Yaskawa INFORM job: R1_W26(-90,90)(KAMERA).JBI

/JOB
//NAME R1_W26(-90,90)(KAMERA)
//POS
///NPOS 78,78,0,7,0,0
///TOOL 0
///POSTYPE PULSE
///PULSE
C00000=-75114,-71893,-86548,-16593,83246,79420
C00001=-80306,-57562,-63247,-15413,75536,78631
C00002=-81645,-55087,-59639,-15080,74370,78302
C00003=-81645,-55006,-58527,-15126,73749,78382
C00004=-81645,-55025,-58760,-15117,73878,78365
C00005=-82615,-56005,-59303,-14838,73537,78058
C00006=-81645,-55079,-59521,-15087,74304,78310
C00007=-93593,1947,-22095,-11058,78527,73697
C00008=-93896,1420,-20145,-11015,77043,73728
C00009=-93896,1359,-19447,-11035,76591,73769
C00010=-93896,1375,-19639,-11030,76716,73757
C00011=-94601,778,-20143,-10801,76623,73523
C00012=-93896,1456,-20502,-11006,77276,73706
C00013=-99701,55982,31111,-9246,72874,72061
C00014=-100041,56496,33717,-9193,71511,72046
C00015=-100041,56569,34702,-9223,70950,72089
C00016=-100041,56551,34487,-9216,71073,72080
C00017=-100636,55976,33841,-9009,71106,71866
C00018=-100041,56488,33604,-9190,71578,72041
C00019=-99543,52569,25332,-9219,74671,71979
C00020=-97259,35030,-12066,-9701,88745,71659
C00021=-112921,-101015,-99029,5314,69459,84771
C00022=-131689,-93265,-75977,27197,64180,77750
C00023=-125720,-68183,-62010,24523,66206,80662
C00024=-125720,-67997,-61190,24597,65833,80578
C00025=-125720,-68044,-61398,24578,65929,80599
C00026=-124863,-68129,-61441,24298,65661,80883
C00027=-125720,-68320,-62645,24468,66502,80726
C00028=-125720,-68684,-64449,24312,67343,80914
C00029=-124059,-8041,-25847,22767,73693,82865
C00030=-124059,-8098,-23570,22924,72370,82603
C00031=-124059,-8098,-23067,22960,72086,82548
C00032=-124059,-8098,-23269,22945,72201,82571
C00033=-123393,-8156,-23316,22717,72018,82785
C00034=-124059,-8088,-24456,22861,72880,82707
C00035=-124059,-8025,-26153,22747,73876,82901
C00036=-123243,49165,27702,22910,70180,82472
C00037=-123243,49353,29898,23083,69020,82237
C00038=-123243,49474,30981,23171,68462,82121
C00039=-123243,49447,30748,23151,68580,82145
C00040=-122653,49389,30685,22948,68426,82342
C00041=-123243,49309,29455,23047,69250,82282
C00042=-123261,47212,24063,22760,71328,82695
C00043=-127182,-101970,-83118,25859,62678,79240
C00044=-148123,-105377,-50787,80405,47389,50643
C00045=-144996,-106265,-51019,81268,45275,50701
C00046=-125639,-92184,-72932,25604,61069,79507
C00047=-125809,-91535,-71625,25772,60696,79344
C00048=-125196,-74812,-64441,24671,64300,80456
C00049=-124580,-57199,-55547,23834,67394,81387
C00050=-124115,-40866,-46002,23300,69579,82027
C00051=-123813,-29133,-38349,23019,70716,82374
C00052=-123561,-15314,-28491,22802,71603,82649
C00053=-123288,-2303,-18230,22666,71872,82806
C00054=-123046,12376,-5585,22611,71586,82839
C00055=-122891,24863,5995,22646,70888,82760
C00056=-122733,39263,20347,22777,69515,82548
C00057=-122600,54559,36695,23052,67446,82176
C00058=-122491,73744,58718,23649,64007,81492
C00059=-122584,71948,49831,22918,68228,82344
C00060=-109861,31401,-26015,2772,95783,84263
C00061=-100600,-80082,-88673,-18141,88148,63436
C00062=-108129,-100882,-75117,-22380,56663,65945
C00063=-110628,-101357,-75286,-21477,55869,65041
C00064=-108411,-101318,-76207,-22166,57003,65749
C00065=-110367,-78057,-70654,-16601,76479,61655
C00066=-111567,-60993,-62345,-16165,79753,60785
C00067=-112558,-45358,-53437,-15865,82017,60140
C00068=-113363,-29494,-43337,-15644,83731,59640
C00069=-113890,-17207,-34628,-15515,84553,59355
C00070=-114365,-3587,-24043,-15417,84933,59146
C00071=-114796,9143,-13275,-15325,84771,59016
C00072=-115137,22513,-1051,-15263,84075,58986
C00073=-115459,35059,11282,-15217,82911,59020
C00074=-115787,51150,28216,-15212,80770,59169
C00075=-116132,68584,47996,-15279,77596,59448
C00076=-116103,68586,47975,-15286,77615,59456
C00077=-116215,70911,26590,-15008,91479,57719
BC00000=318604,15,1075175
BC00001=318604,15,1075175
BC00002=318604,15,1075175
BC00003=318604,15,1075175
BC00004=318604,15,1075175
BC00005=318604,15,1075175
BC00006=318604,15,1075175
BC00007=318604,15,1075175
BC00008=318604,15,1075175
BC00009=318604,15,1075175
BC00010=318604,15,1075175
BC00011=318604,15,1075175
BC00012=318604,15,1075175
BC00013=318604,15,1075175
BC00014=318604,15,1075175
BC00015=318604,15,1075175
BC00016=318604,15,1075175
BC00017=318604,15,1075175
BC00018=318604,15,1075175
BC00019=318604,15,1075175
BC00020=318604,15,1075175
BC00021=23891,15,1075175
BC00022=23891,15,1075175
BC00023=23891,15,1075175
BC00024=23891,15,1075175
BC00025=23891,15,1075175
BC00026=23891,15,1075175
BC00027=23891,15,1075175
BC00028=23891,15,1075175
BC00029=23891,15,1075175
BC00030=23891,15,1075175
BC00031=23891,15,1075175
BC00032=23891,15,1075175
BC00033=23891,15,1075175
BC00034=23891,15,1075175
BC00035=23891,15,1075175
BC00036=23891,15,1075175
BC00037=23891,15,1075175
BC00038=23891,15,1075175
BC00039=23891,15,1075175
BC00040=23891,15,1075175
BC00041=23891,15,1075175
BC00042=23891,15,1075175
BC00043=23891,15,1075175
BC00044=23891,15,1075175
BC00045=23891,15,1075175
BC00046=23891,15,1075175
BC00047=23891,15,1075175
BC00048=23891,15,1075175
BC00049=23891,15,1075175
BC00050=23891,15,1075175
BC00051=23891,15,1075175
BC00052=23891,15,1075175
BC00053=23891,15,1075175
BC00054=23891,15,1075175
BC00055=23891,15,1075175
BC00056=23891,15,1075175
BC00057=23891,15,1075175
BC00058=23891,15,1075175
BC00059=23891,15,1075175
BC00060=194351,494,1075175
BC00061=393793,1055,1075176
BC00062=393793,1055,1075176
BC00063=393793,1055,1075176
BC00064=393793,1055,1075176
BC00065=393793,1055,1075176
BC00066=393793,1053,1075174
BC00067=393793,1053,1075174
BC00068=393793,1053,1075174
BC00069=393793,1053,1075174
BC00070=393793,1053,1075172
BC00071=393793,1053,1075172
BC00072=393793,1053,1075172
BC00073=393793,1053,1075172
BC00074=393793,1053,1075172
BC00075=393793,1053,1075172
BC00076=393793,17497,1075172
BC00077=393793,17497,1075172
///POSTYPE BASE
///RECTAN
///RCONF 0,0,0,0,1,0,0,0,0,0,0,0,0,0,0,0,0,0,0,0,0,0,0,0
P00006=2.006,1.622,-0.565,0.0000,0.0000,0.0000
P00021=0.073,2.058,-0.109,0.0000,0.0000,0.0000
P00022=2.006,1.622,-0.565,0.0000,0.0000,0.0000
///RCONF 0,0,0,0,0,0,0,0,0,0,0,0,0,0,0,0,0,0,0,0,0,0,0,0
P00023=-2.957,-4.083,2.762,0.0000,0.0000,0.0000
P00024=-1.466,-0.226,-0.419,0.0000,0.0000,0.0000
P00025=3.643,0.007,-2.585,0.0000,0.0000,0.0000
P00026=2.644,0.055,-2.583,0.0000,0.0000,0.0000
//INST
///DATE 2025/04/11 09:13
///ATTR SC,RW
///GROUP1 RB1,BS1
NOP
SFTOF
CALL JOB:ONLYCUT-R1_LONG
SFTOF
MOVJ C00000 BC00000 VJ=100.00
MOVJ C00001 BC00001 VJ=100.00
'P1
MOVL C00002 BC00002 V=133.3
REFP 3 C00003 BC00003
CALL JOB:SEARCH-R1
SET P021 P006
SFTON P021
MOVL C00004 BC00004 V=66.7
REFP 3 C00005 BC00005
CALL JOB:SEARCH-R1
SET P021 P006
SFTON P021
MOVL C00006 BC00006 V=133.3
SFTOF
MOVL C00007 BC00007 V=1000.0
'P2
MOVL C00008 BC00008 V=133.3
REFP 3 C00009 BC00009
CALL JOB:SEARCH-R1
SET P022 P006
SFTON P022
MOVL C00010 BC00010 V=66.7
REFP 3 C00011 BC00011
CALL JOB:SEARCH-R1
SET P022 P006
SFTON P022
MOVL C00012 BC00012 V=133.3
SFTOF
MOVL C00013 BC00013 V=1000.0
'P3
MOVL C00014 BC00014 V=133.3
REFP 3 C00015 BC00015
CALL JOB:SEARCH-R1
SET P023 P006
SFTON P023
MOVL C00016 BC00016 V=83.3
REFP 3 C00017 BC00017
CALL JOB:SEARCH-R1
SET P023 P006
SFTON P023
MOVL C00018 BC00018 V=133.3
SFTOF
MOVL C00019 BC00019 V=1000.0
MOVJ C00020 BC00020 VJ=100.00
MOVJ C00021 BC00021 VJ=100.00
MOVJ C00022 BC00022 VJ=100.00
MOVL C00023 BC00023 V=133.3
'P1
REFP 3 C00024 BC00024
CALL JOB:SEARCH-R1
SET P024 P006
SFTON P024
MOVL C00025 BC00025 V=66.7
REFP 3 C00026 BC00026
CALL JOB:SEARCH-R1
SET P024 P006
SFTON P024
MOVL C00027 BC00027 V=133.3
SFTOF
MOVL C00028 BC00028 V=333.3
MOVL C00029 BC00029 V=1000.0
MOVL C00030 BC00030 V=133.3
'P2
REFP 3 C00031 BC00031
CALL JOB:SEARCH-R1
SET P025 P006
SFTON P025
MOVL C00032 BC00032 V=66.7
REFP 3 C00033 BC00033
CALL JOB:SEARCH-R1
SET P025 P006
SFTON P025
MOVL C00034 BC00034 V=133.3
SFTOF
MOVL C00035 BC00035 V=333.3
MOVL C00036 BC00036 V=333.3
MOVL C00037 BC00037 V=133.3
'P3
REFP 3 C00038 BC00038
CALL JOB:SEARCH-R1
SET P026 P006
SFTON P026
MOVL C00039 BC00039 V=66.7
REFP 3 C00040 BC00040
CALL JOB:SEARCH-R1
SET P026 P006
SFTON P026
MOVL C00041 BC00041 V=133.3
SFTOF
CALL JOB:COFNIJ_DRUT
MOVL C00042 BC00042 V=333.3
MOVL C00043 BC00043 V=1000.0
MACRO1 MJ#(0) ARGF9
SFTON P024
MOVJ C00044 BC00044 VJ=25.00
ARCON
MOVL C00045 BC00045 V=11.0
ARCOF
MOVJ C00046 BC00046 VJ=25.00
MOVJ C00047 BC00047 VJ=15.00
MACRO1 MJ#(0) ARGF9
ARCON
MOVL C00048 BC00048 V=13.3
ARCOF
MOVL C00049 BC00049 V=41.7
ARCON
MOVL C00050 BC00050 V=13.3
ARCOF
SFTOF
SFTON P025
MOVL C00051 BC00051 V=83.3
ARCON
MOVL C00052 BC00052 V=13.3
ARCOF
MOVL C00053 BC00053 V=83.3
ARCON
MOVL C00054 BC00054 V=13.3
ARCOF
SFTOF
SFTON P026
MOVL C00055 BC00055 V=83.3
ARCON
MOVL C00056 BC00056 V=13.3
ARCOF
MOVL C00057 BC00057 V=83.3
ARCON
MOVL C00058 BC00058 V=16.7
ARCOF
MOVL C00059 BC00059 V=166.7
MOVJ C00060 BC00060 VJ=100.00
MOVJ C00061 BC00061 VJ=100.00
SFTON P021
MOVJ C00062 BC00062 VJ=25.00
ARCON
MOVL C00063 BC00063 V=11.0
ARCOF
MOVL C00064 BC00064 V=83.3
MOVL C00065 BC00065 V=166.7
ARCON
MOVL C00066 BC00066 V=13.3
ARCOF
MOVL C00067 BC00067 V=83.3
ARCON
MOVL C00068 BC00068 V=13.3
ARCOF
SFTOF
SFTON P022
MOVL C00069 BC00069 V=83.3
ARCON
MOVL C00070 BC00070 V=13.3
ARCOF
MOVL C00071 BC00071 V=83.3
ARCON
MOVL C00072 BC00072 V=13.3
ARCOF
SFTOF
SFTON P023
MOVL C00073 BC00073 V=83.3
ARCON
MOVL C00074 BC00074 V=13.3
ARCOF
MOVL C00075 BC00075 V=83.3
ARCON
MOVL C00076 BC00076 V=16.7
ARCOF
SFTOF
MOVL C00077 BC00077 V=166.7
END
